(* PLC project Generated.project, CODESYS CODESYS V3.5 SP19 Patch 1 *)
(* stored: creationDateTime 2026-08-18T12:52:51.260137, modificationDateTime 2026-08-18T12:52:51.260137 *)

TYPE ST_Chain_Winch_Control : STRUCT
  Idx401_MotionAllowed : BOOL;  (* 1 = Prêt / Mouvement Autorisé | 0 = Bloqué *)
  Idx402_SpeedStepCalculated : INT;  (* Palier Vitesse Calculé (0, 1, 2, 3, 4) *)
  Idx403_SpeedRamp_Pct : REAL;  (* [%] Consigne Vitesse après Rampe *)
  Idx404_BrakeReleaseAuthorized : BOOL;  (* 1 = Ordre Ouverture Frein | 0 = Ordre Serrage *)
  Idx405_FinalInterlockState : E_WinchFinalInterlockState;  (* 🛡️ État frontière _LD *)
  Idx406_FinalInterlockReason : E_WinchFinalInterlockReason;  (* 🛡️ Cause mémorisée *)
  Idx407_FinalAuthorizedStep : INT;  (* 🪜 Palier réellement autorisé *)
  Idx408_BrakeCommandOpenConfirmed : BOOL;  (* 🔌 Contacteur/bobine, pas frein mécanique *)
  Idx409_BrakeTimeoutElapsed : TIME;  (* ⏱️ Watchdog 500ms écoulé *)
  Idx410_RestartDelayElapsed : TIME;  (* ⏱️ Verrou 900ms écoulé *)
  Idx411_StepDelayElapsed : TIME;  (* ⏱️ Délai palier 1s250 écoulé *)
  Idx412_InTopSlowdownZone : BOOL;  (* : Palier plafonné à 1, approche limite haute *)
  Idx413_InBottomSlowdownZone : BOOL;  (* : Palier plafonné à 1, approche limite basse (câble ou légale) *)
  Idx414_BottomLimitActiveM : REAL;  (* : Limite basse active (m) — câble physique OU légale, la plus restrictive *)
END_STRUCT;
END_TYPE

(* values of E_WinchFinalInterlockReason: NONE: Aucun blocage actif; BRAKE_COMMAND_NOT_CONFIRMED: Absence confirmation ouverture frein > 500ms; RESTART_INHIBITED: Inhibition redemarrage actif *)

{attribute 'qualified_only'}
{attribute 'strict'}
TYPE E_WinchFinalInterlockReason : (NONE := 0, BRAKE_COMMAND_NOT_CONFIRMED := 1, RESTART_INHIBITED := 2);
END_TYPE

(* values of E_WinchFinalInterlockState: DISABLED: Desactive / Hors service; READY: Pret / Etat nominal; WAIT_BRAKE_COMMAND_CONFIRMATION: Attente confirmation feedback frein; WAIT_STEP_DELAY: Temporisation changement de palier; WAIT_RESTART_DELAY: Temporisation anti-court-cycle redemarrage; FAULT: Etat de defaut *)

{attribute 'qualified_only'}
{attribute 'strict'}
TYPE E_WinchFinalInterlockState : (DISABLED := 0, READY := 1, WAIT_BRAKE_COMMAND_CONFIRMATION := 2, WAIT_STEP_DELAY := 3, WAIT_RESTART_DELAY := 4, FAULT := 5);
END_TYPE
